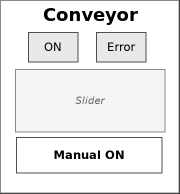
VISUALIZATION vConveyor  // 180x194
VAR_INPUT
	iNameIndex :INT;
END_VAR
VAR_IN_OUT
	fbConveyor :FB_Conveyor;

END_VAR
    Rectangle (0,0 180x194)
    Rectangle (28,32 50x30), "ON", colour toggle: fbConveyor.prIsOn
    Rectangle (35,0 111x30), "Conveyor", text list: 'tlDevices', text index: iNameIndex
    Rectangle (96,32 50x30), "Error", colour toggle: fbConveyor.prError
    Rectangle (16,137 146x36), "Manual ON", colour toggle: fbConveyor.bManualOnCmd, input disabled if: NOT fbConveyor.bManualMode
        toggle fbConveyor.bManualOnCmd
    Slider (15,69 150x63), variable: fbConveyor.rSpeedSet, scale 0..100
END_VISUALIZATION

(* stored: Version 1.1.0.1, ProductVersion 3.1.4024.15
   Visu vConveyor: Id {3d896d0c-fc0d-4a44-b6c7-bb98fb0d3294} *)
